FUNCTION_BLOCK CAerationSensors (* Composite Function Block Type *)
  (* Standard: 61499-2 *)
  (* Version 0.0, 7/1/2024, NVPP, Schneider Electric, template *)
  PACKAGE SE.Nereda;
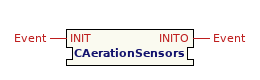
  EVENT_INPUT
    INIT;
  END_EVENT
  EVENT_OUTPUT
    INITO;
  END_EVENT
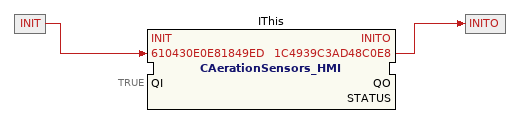
  (* 01 - FUNCTIONNAL INPUT INTERFACE *)
  (* 00 - INITIALIZATION *)
  (* 06 - HMI INTERFACE *)
  (* 02 - FUNCTIONNAL OUTPUT INTERFACE *)
  (* 03 - FIELD INTERFACE *)
  FBS
    IThis : CAerationSensors_HMI(QI := TRUE);
  END_FBS
  EVENT_CONNECTIONS
    INIT TO IThis.610430E0E81849ED;
    IThis.1C4939C3AD48C0E8 TO INITO;
  END_CONNECTIONS
END_FUNCTION_BLOCK
